{attribute 'qualified_only'}
VAR_GLOBAL CONSTANT
	MaxAmountObject				: UINT := 10000;
END_VAR

(* stored: Version 1.1.0.1
   GVL Par_InitManager: Id {0e81be1d-468a-4f8b-a2f4-876f05071527}, ParameterList True *)
